// TIA Portal V18 export
FUNCTION_BLOCK "FB23-regenarationpgmFB"   // FB23, LAD
{ S7_Optimized_Access := 'TRUE' }
VERSION : 0.1
// stored: AutoNumber false, IsIECCheckEnabled false, IsRetainMemResEnabled false, MemoryReserve 100, SetENOAutomatically false, UDAEnableTagReadback false
   VAR_INPUT
      Dispensing_time : DInt;
      "Set Qty in ml" : Real;
      "Pump ON A delay" : DInt;
      "Pump ON B delay" : DInt;
      "Mixer Off delay" : DInt;
   END_VAR
   VAR_OUTPUT
      "Run time" : Int;
   END_VAR
   VAR_IN_OUT
      ON_Pump_A : Bool;
      ON_pump_B : Bool;
      ON_Mixer : Bool;
      "Start Metering" : Bool;
      "Stop metering" : Bool;
      "Process running" : Bool;
      "process completed" : Bool;
   END_VAR
   VAR
      "Total Volume dispensed" : Real;
      "metering started" : Bool;
      "metering time in msec" : DInt;
      "dispense time elapsed" : Bool;
   END_VAR
   VAR_TEMP
      Ons_temp : Bool;
   END_VAR
   VAR_TEMP   // added for the SCL form of the ladder/FBD networks
      _w1 : Bool;
   END_VAR
BEGIN

REGION Network 1
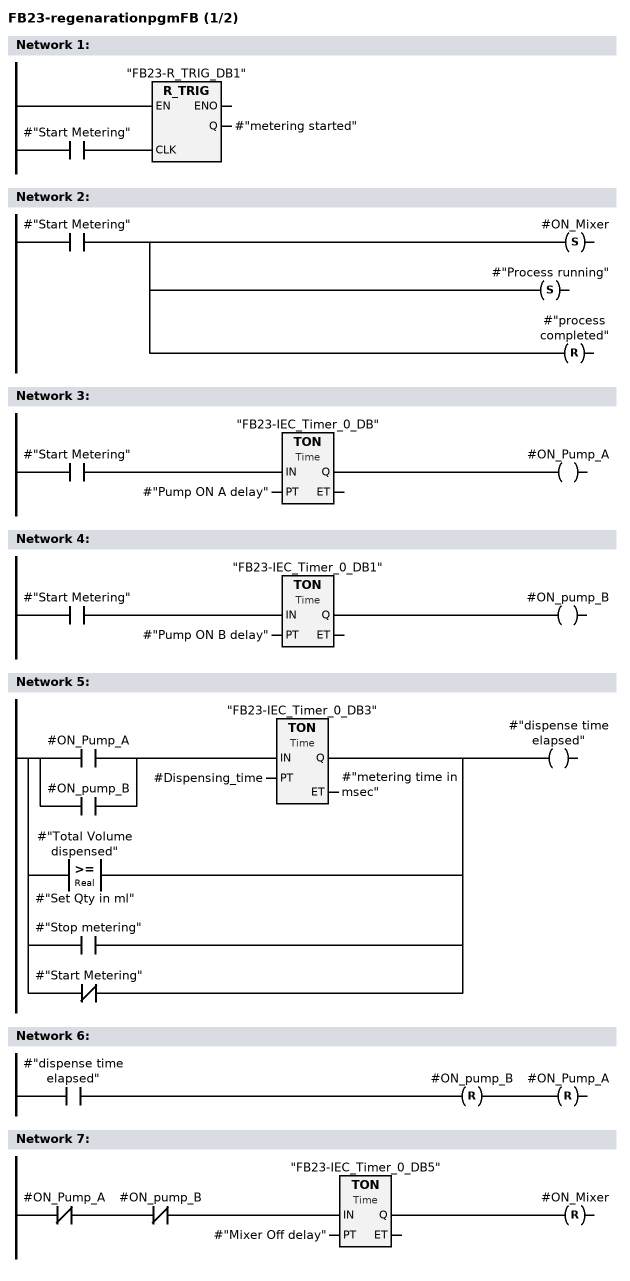
   RUNG wire#powerrail
      "FB23-R_TRIG_DB1".R_TRIG(CLK := wire#w1, Q => #"metering started")
   END_RUNG
   RUNG wire#powerrail
      Contact( #"Start Metering" )
   END_RUNG wire#w1
   // the same network as SCL:
   "FB23-R_TRIG_DB1"(CLK := #"Start Metering", Q => #"metering started");   // R_TRIG
END_REGION

REGION Network 2
   RUNG wire#powerrail
      Contact( #"Start Metering" )
      wire#w1
      S_Coil( #ON_Mixer )
   END_RUNG
   RUNG wire#w1
      S_Coil( #"Process running" )
   END_RUNG
   RUNG wire#w1
      R_Coil( #"process completed" )
   END_RUNG
   // the same network as SCL:
   IF #"Start Metering" THEN
       #ON_Mixer := TRUE;
       #"Process running" := TRUE;
       #"process completed" := FALSE;
   END_IF;
END_REGION

REGION Network 3
   RUNG wire#powerrail
      Contact( #"Start Metering" )
      { S7_Templates := "time_type := Time" } "FB23-IEC_Timer_0_DB".TON(pt := #"Pump ON A delay", et =>)
      Coil( #ON_Pump_A )
   END_RUNG
   // the same network as SCL:
   "FB23-IEC_Timer_0_DB".TON(IN := #"Start Metering", PT := #"Pump ON A delay");
   #ON_Pump_A := "FB23-IEC_Timer_0_DB".Q;
END_REGION

REGION Network 4
   RUNG wire#powerrail
      Contact( #"Start Metering" )
      { S7_Templates := "time_type := Time" } "FB23-IEC_Timer_0_DB1".TON(pt := #"Pump ON B delay", et =>)
      Coil( #ON_pump_B )
   END_RUNG
   // the same network as SCL:
   "FB23-IEC_Timer_0_DB1".TON(IN := #"Start Metering", PT := #"Pump ON B delay");
   #ON_pump_B := "FB23-IEC_Timer_0_DB1".Q;
END_REGION

REGION Network 5
   RUNG wire#powerrail
      Contact( #ON_Pump_A )
      wire#w1
      { S7_Templates := "time_type := Time" } "FB23-IEC_Timer_0_DB3".TON(pt := #Dispensing_time, et => #"metering time in msec")
      wire#w2
      Coil( #"dispense time elapsed" )
   END_RUNG
   RUNG wire#powerrail
      Contact( #ON_pump_B )
   END_RUNG wire#w1
   RUNG wire#powerrail
      { S7_Templates := "SrcType := Real" } GE_Contact(in1 := #"Total Volume dispensed", in2 := #"Set Qty in ml")
   END_RUNG wire#w2
   RUNG wire#powerrail
      Contact( #"Stop metering" )
   END_RUNG wire#w2
   RUNG wire#powerrail
      I_Contact( #"Start Metering" )
   END_RUNG wire#w2
   // the same network as SCL:
   "FB23-IEC_Timer_0_DB3".TON(IN := #ON_Pump_A OR #ON_pump_B,
                           PT := #Dispensing_time,
                           ET => #"metering time in msec");
   #"dispense time elapsed" := "FB23-IEC_Timer_0_DB3".Q OR (#"Total Volume dispensed" >= #"Set Qty in ml") OR #"Stop metering" OR NOT #"Start Metering";
END_REGION

REGION Network 6
   RUNG wire#powerrail
      Contact( #"dispense time elapsed" )
      R_Coil( #ON_pump_B )
      R_Coil( #ON_Pump_A )
   END_RUNG
   // the same network as SCL:
   IF #"dispense time elapsed" THEN
       #ON_pump_B := FALSE;
       #ON_Pump_A := FALSE;
   END_IF;
END_REGION

REGION Network 7
   RUNG wire#powerrail
      I_Contact( #ON_Pump_A )
      I_Contact( #ON_pump_B )
      { S7_Templates := "time_type := Time" } "FB23-IEC_Timer_0_DB5".TON(pt := #"Mixer Off delay", et =>)
      R_Coil( #ON_Mixer )
   END_RUNG
   // the same network as SCL:
   "FB23-IEC_Timer_0_DB5".TON(IN := NOT #ON_Pump_A AND NOT #ON_pump_B, PT := #"Mixer Off delay");
   IF "FB23-IEC_Timer_0_DB5".Q THEN #ON_Mixer := FALSE; END_IF;
END_REGION

REGION Network 8
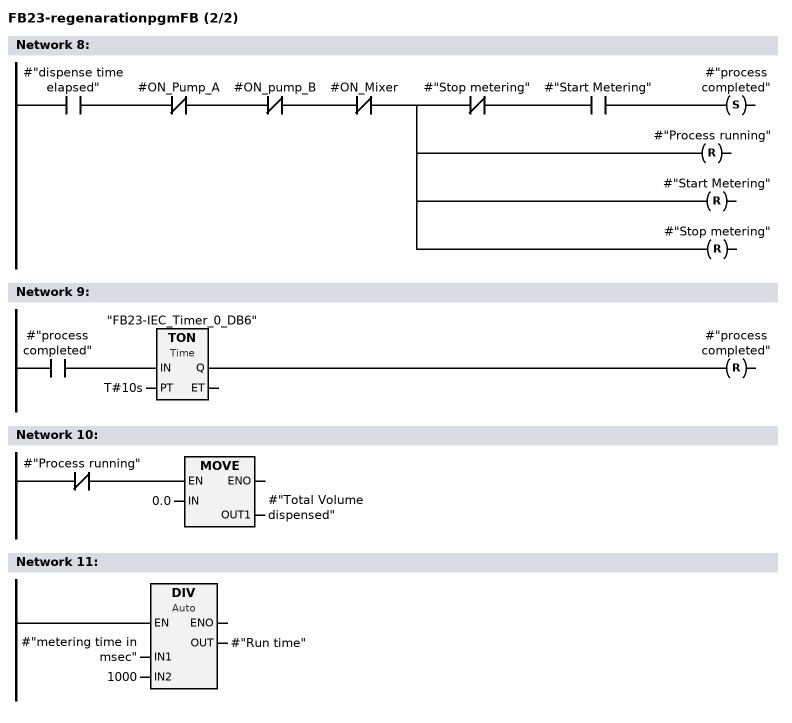
   RUNG wire#powerrail
      Contact( #"dispense time elapsed" )
      I_Contact( #ON_Pump_A )
      I_Contact( #ON_pump_B )
      I_Contact( #ON_Mixer )
      wire#w1
      I_Contact( #"Stop metering" )
      Contact( #"Start Metering" )
      S_Coil( #"process completed" )
   END_RUNG
   RUNG wire#w1
      R_Coil( #"Process running" )
   END_RUNG
   RUNG wire#w1
      R_Coil( #"Start Metering" )
   END_RUNG
   RUNG wire#w1
      R_Coil( #"Stop metering" )
   END_RUNG
   // the same network as SCL:
   #_w1 := #"dispense time elapsed" AND NOT #ON_Pump_A AND NOT #ON_pump_B AND NOT #ON_Mixer;
   IF #_w1 AND NOT #"Stop metering" AND #"Start Metering" THEN #"process completed" := TRUE; END_IF;
   IF #_w1 THEN
       #"Process running" := FALSE;
       #"Start Metering" := FALSE;
       #"Stop metering" := FALSE;
   END_IF;
END_REGION

REGION Network 9
   RUNG wire#powerrail
      Contact( #"process completed" )
      { S7_Templates := "time_type := Time" } "FB23-IEC_Timer_0_DB6".TON(pt := T#10s, et =>)
      R_Coil( #"process completed" )
   END_RUNG
   // the same network as SCL:
   "FB23-IEC_Timer_0_DB6".TON(IN := #"process completed", PT := T#10s);
   IF "FB23-IEC_Timer_0_DB6".Q THEN #"process completed" := FALSE; END_IF;
END_REGION

REGION Network 10
   RUNG wire#powerrail
      I_Contact( #"Process running" )
      Move(in := 0.0, out1 => #"Total Volume dispensed")
   END_RUNG
   // the same network as SCL:
   IF NOT #"Process running" THEN #"Total Volume dispensed" := 0.0; END_IF;
END_REGION

REGION Network 11
   RUNG wire#powerrail
      Div(in1 := #"metering time in msec", in2 := 1000, out => #"Run time")
   END_RUNG
   // the same network as SCL:
   #"Run time" := #"metering time in msec" / 1000;
END_REGION
END_FUNCTION_BLOCK
